Fanuc KAREL source: kd00050.KL

-- PROVISIONAL review KL for V1013-1; original PC SHA256 73273ee4223bf908425990f29242c6ac7cd26dfebb78d3be7f0453a8f4050392
-- Incomplete behavior may be omitted. Consult companion uncertainty JSON. Do not deploy.
PROGRAM KD00050
%NOLOCKGROUP
VAR
  I : INTEGER
  J : INTEGER
  B : BOOLEAN
  R : REAL
  S : STRING[80]
BEGIN
  -- UNRESOLVED_PC offsets 5-19; opcodes 01,9D,2E,0A,82,0B
  -- UNRESOLVED_PC offsets 24-28; opcodes 7F
END KD00050
